{attribute 'qualified_only'}
VAR_GLOBAL
	stVirtualInputs : ST_VirtualInputs;
	stVirtualOutputs : ST_VirtualOutputs;
END_VAR

(* stored: Version 1.1.0.1, ProductVersion 3.1.4024.9
   GVL VirtualControlBox: Id {0ca5c0a4-0d20-4ce5-afdb-fe579593098c} *)
